(* Schneider Machine Expert - Basic project Contador, file version 2.7.0.0 *)
(* ProjectInformations: Name=Nuevo proyecto *)

HARDWARE
  Cpu 0: TM221M16R/G
  ModuleExtensionObject 0: TM3DI16K
  EthernetConfiguration: NetworkName=M221, IpAllocationMode=FixedAddress, IpAddress=0.0.0.0, SubnetMask=0.0.0.0
  SerialLineConfiguration: Baud=Baud19200, Parity=ParityEven, DataBits=DataBits8, StopBits=StopBits1, PhysicalMedium=PhysicalMediumRs485, TransmissionMode=TransmissionModeModbusRtu, SlaveId=1, Addressing=SlaveAddressing
  MastTask: UsePeriodScanMode=false, PeriodScan=100
  FastTask: Period=255
  CpuBehavior: StartingMode=StartAsPreviousState, AutoSaveRamOnEeprom=true, WatchdogPeriod=250

SYMBOLS  (address, symbol, comment, settings)
  %M1         "At Entry"
  %M2         "At Exit"
  %M4         "Entry Conveyor"
  %M5         "Exit Conveyor"
  %M100       "Active"
  %M101       "Auxiliar"
  %C0         "Contador"  [Preset=3]

POU Nuevo POU
  (* SectionNumber=1 *)

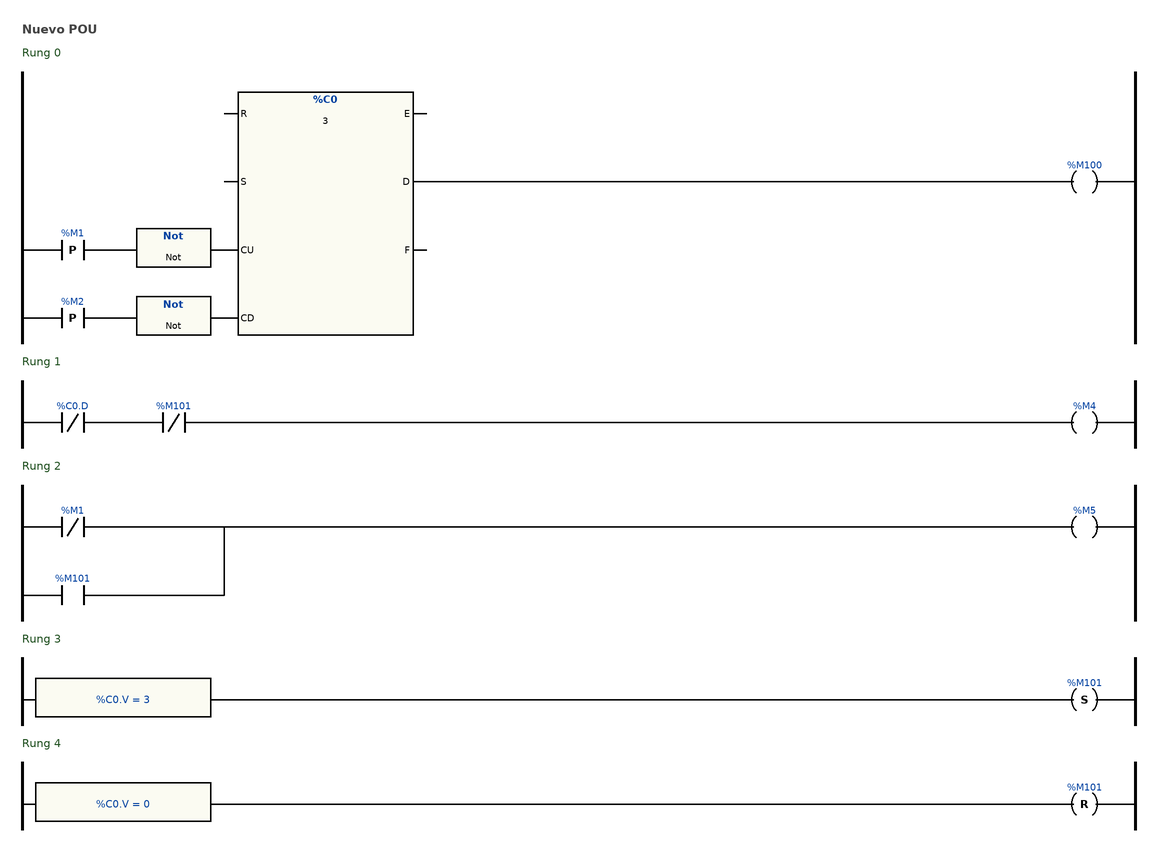

// Rung 0
  BLK %C0
  LDR %M1
  N
  CU
  LDR %M2
  N
  CD
  OUT_BLK
  LD D
  ST %M100
  END_BLK
  // as ST:
  //   %C0(CU := NOT RISING(%M1), CD := NOT RISING(%M2));
  //   %M100 := %C0.D;

// Rung 1
  LDN %C0.D
  ANDN %M101
  ST %M4
  // as ST:
  //   %M4 := NOT %C0.D AND NOT %M101;

// Rung 2
  LDN %M1
  OR %M101
  ST %M5
  // as ST:
  //   %M5 := NOT %M1 OR %M101;

// Rung 3
  LD [ %C0.V = 3 ]
  S %M101
  // as ST:
  //   IF %C0.V = 3 THEN %M101 := TRUE; END_IF;

// Rung 4
  LD [ %C0.V = 0 ]
  R %M101
  // as ST:
  //   IF %C0.V = 0 THEN %M101 := FALSE; END_IF;
